TEXTLIST TextList_Util_Group
  1 = 'Liste des groupes' | FR: 'Liste des groupes' | EN: 'Group list'
  3 = 'Edition procédés' | FR: 'Edition procédés' | EN: 'Process edition'
  4 = 'Maintenance' | FR: 'Maintenance' | EN: 'Maintenance'
  5 = 'Administrateur' | FR: 'Administrateur' | EN: 'Administrator'
  6 = 'Production' | FR: 'Production' | EN: 'Production'
  7 = 'Configuration' | FR: 'Configuration' | EN: 'Settings'
  8 = 'Fonctions avancées' | FR: 'Fonctions avancées' | EN: 'Advanced functions'
  9 = 'Modif groupe' | FR: 'Modification du groupe' | EN: 'Group modification'
  10 = 'Creation groupe' | FR: "Création d'un groupe" | EN: 'Group creation'
   = ''
END_TEXTLIST

(* stored: Version 1.1.0.1, ProductVersion 3.1.4024.10
   TextList TextList_Util_Group: Id {dc107d42-fa29-4400-8e39-aa81e20d6b3a} *)
